INTERFACE I_ContinuousDrive EXTENDS I_Drive

METHOD ABSTRACT moveContinuous : BOOL
VAR_INPUT
	direction : MC_Direction;
END_VAR
END_METHOD

END_INTERFACE

(* stored: Version 1.1.0.1, ProductVersion 3.1.4024.11
   Itf I_ContinuousDrive: Id {e0e763c8-82fe-4e71-b666-b1f5372719c5}
   Method moveContinuous: Id {06e4620f-ea1c-43d6-b81a-6ac6275bc821} *)
